PROGRAM MAIN
VAR
END_VAR

END_PROGRAM

(* stored: Version 1.1.0.1
   POU MAIN: Id {60cb77d4-9ad5-4845-a91a-5fcb5ee5d0f3} *)
